# EPICS autosave request: ADApp/Db/ADAutoSaveMenu.req
file "configMenu.req", P=$(P), CONFIG=ADAutoSave
file "auto_settings.req", P=$(P)
